INTERFACE IPmlStateMachine

METHOD GetCurrentState : E_PMLState
VAR_INPUT
END_VAR
END_METHOD

METHOD PMLCommand : bool
VAR_INPUT
	Command : E_PMLCommand;
END_VAR
END_METHOD

METHOD StateComplete : BOOL
VAR_INPUT
END_VAR
END_METHOD

END_INTERFACE

(* stored: Version 1.1.0.1, ProductVersion 3.1.4024.11
   Itf IPmlStateMachine: Id {a572c756-2ee2-4617-b1ba-a370e2347b9e}
   Method GetCurrentState: Id {8896b180-4065-4462-9182-dfc33f7be59c}
   Method PMLCommand: Id {f841f4da-d94f-47fd-a3c7-c8897a849506}
   Method StateComplete: Id {5723ee2f-d368-4970-a6c6-2e134230c395} *)
